% RSLogix 500 project EXCER_BAK060.RSS, saved by version 8.10.00.18 %
PROJECT "UNTITLED"    % processor: MicroLogix 1200 %

PROGRAM FILES
  LAD 2   7 rungs

DATA FILES
  O0 OUTPUT  4 elements
  I1 INPUT  4 elements
  S2 STATUS  66 elements
  B3 BINARY  1 elements
  T4 TIMER  1 elements
  C5 COUNTER  1 elements
  R6 CONTROL  1 elements
  N7 INTEGER  1 elements

LADDER 2
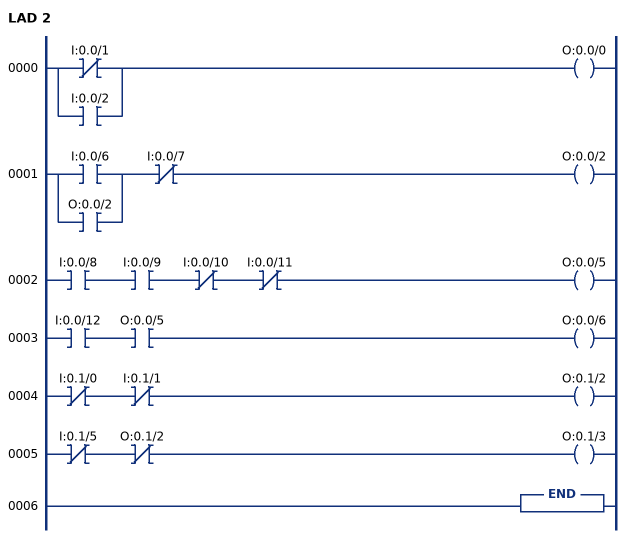
% Rung: 0 %
SOR BST XIO I:0.0/1 NXB XIC I:0.0/2 BND OTE O:0.0/0 EOR
% Rung: 1 %
SOR BST XIC I:0.0/6 NXB XIC O:0.0/2 BND XIO I:0.0/7 OTE O:0.0/2 EOR
% Rung: 2 %
SOR XIC I:0.0/8 XIC I:0.0/9 XIO I:0.0/10 XIO I:0.0/11 OTE O:0.0/5 EOR
% Rung: 3 %
SOR XIC I:0.0/12 XIC O:0.0/5 OTE O:0.0/6 EOR
% Rung: 4 %
SOR XIO I:0.1/0 XIO I:0.1/1 OTE O:0.1/2 EOR
% Rung: 5 %
SOR XIO I:0.1/5 XIO O:0.1/2 OTE O:0.1/3 EOR
% Rung: 6 %
SOR END EOR
